TYPE PROG_STEPS :
STRUCT

	VAC_STEP:INT;
	Q1_STEP:INT;
	Q2_STEP:INT;
	PMAX_STEP:INT;
	PRINT_STEP:INT;


END_STRUCT
END_TYPE

(* stored: Version 1.1.0.1, ProductVersion 3.1.0.26
   DUT PROG_STEPS: Id {3527081a-deb7-4f80-9971-0053b3b68c31} *)
